// TwinCAT 3 PLC project Untitled1
// ProgramVersion: 3.1.4024.0
// libraries:
//   Tc2_Standard, * (Beckhoff Automation GmbH)
//   Tc2_System, * (Beckhoff Automation GmbH)
//   Tc3_Module, * (Beckhoff Automation GmbH)
// project tree:
//   DUTs/ E_MsMode.TcDUT, ST_ToolBay.TcDUT
//   GVLs/ EMSensor.TcGVL, GVL_Surgeon.TcGVL
//   / PlcTask.TcTTO
//   POUs/ MAIN.TcPOU
//   POUs/S_E_Class/ S_EMSensorPose.TcDUT, ST_EMAdsInput.TcDUT, ST_EMAdsOutput.TcDUT
// real-time tasks:
//   TASK PlcTask: cycle T#10ms, priority 20, ADS port 350

CONFIGURATION Untitled1
    RESOURCE PLC ON TwinCAT3
        TASK PlcTask(INTERVAL := T#10ms, PRIORITY := 20);
        PROGRAM MAIN WITH PlcTask : MAIN;
    END_RESOURCE
END_CONFIGURATION

// ---- DUTs/E_MsMode.TcDUT
{attribute 'strict'}
TYPE E_MsMode :
(
	eMsReleased := 0,	(* 主从释放：屏幕可操作 *)
	eMsPaired   := 1	(* 主从锁定：屏幕锁定，需用户解锁 *)
);
END_TYPE

// ---- DUTs/ST_ToolBay.TcDUT
{attribute 'pack_mode' := '1'}
TYPE ST_ToolBay :
STRUCT
	bToolPresent		: BOOL;	(* 器械在位 *)
	bIsolatorPresent	: BOOL;	(* 隔离板在位；器械在位时必须为 TRUE *)
END_STRUCT
END_TYPE

// ---- POUs/S_E_Class/S_EMSensorPose.TcDUT
{attribute 'pack_mode' := '1'}
TYPE S_EMSensorPose :
STRUCT
	lQuaternion 				: ARRAY[0..3] OF LREAL; // q0, qx, qy, qz
    lPos 						: ARRAY[0..2] OF LREAL; // X, Y, Z，单位 mm
END_STRUCT
END_TYPE

// ---- POUs/S_E_Class/ST_EMAdsInput.TcDUT
{attribute 'pack_mode' := '1'}
TYPE ST_EMAdsInput :
STRUCT
	sEMSensorPose				: ARRAY[1..4] OF S_EMSensorPose; // 下标=NDI通道号，未接入的通道为 0
    lError 						: LREAL;
    lDataScope 					: LREAL;
	bHeatBeat					: BOOL;// 心跳
END_STRUCT
END_TYPE

// ---- POUs/S_E_Class/ST_EMAdsOutput.TcDUT
{attribute 'pack_mode' := '1'}
TYPE ST_EMAdsOutput :
STRUCT
	lDataScope						: ARRAY[0..11] OF LREAL;// 示波器变量
	bHeatBeat						: BOOL;// 心跳
END_STRUCT
END_TYPE

// ---- GVLs/EMSensor.TcGVL
{attribute 'qualified_only'}
{attribute 'pack_mode' := '1'}
VAR_GLOBAL
			stAdsInput  AT%I* : ST_EMAdsInput;
			stAdsOutput AT%Q* : ST_EMAdsOutput;
END_VAR

// ---- GVLs/GVL_Surgeon.TcGVL
{attribute 'qualified_only'}
{attribute 'pack_mode' := '1'}
VAR_GLOBAL
	(* 0=左器械 1=内镜 2=右器械 *)
	arrToolBay		: ARRAY[0..2] OF ST_ToolBay;
	eMsMode			: E_MsMode := E_MsMode.eMsReleased;
	bUserUnlock		: BOOL;	(* HMI → PLC 解锁请求，处理后由 MAIN 清零 *)
END_VAR

// ---- POUs/MAIN.TcPOU
PROGRAM MAIN
VAR
	bInit	: BOOL;
	i		: INT;
END_VAR

IF NOT bInit THEN
	FOR i := 0 TO 2 DO
		GVL_Surgeon.arrToolBay[i].bToolPresent := TRUE;
		GVL_Surgeon.arrToolBay[i].bIsolatorPresent := TRUE;
	END_FOR
	GVL_Surgeon.eMsMode := E_MsMode.eMsReleased;
	bInit := TRUE;
END_IF

(* 医生控制台解锁：收到 HMI 标志后释放主从锁定 *)
IF GVL_Surgeon.bUserUnlock THEN
	GVL_Surgeon.eMsMode := E_MsMode.eMsReleased;
	GVL_Surgeon.bUserUnlock := FALSE;
END_IF

(* 规则：器械在位 ⇒ 隔离板必在位 *)
FOR i := 0 TO 2 DO
	IF GVL_Surgeon.arrToolBay[i].bToolPresent THEN
		GVL_Surgeon.arrToolBay[i].bIsolatorPresent := TRUE;
	END_IF
END_FOR

END_PROGRAM
